// TIA Portal V17 export
// export: Created 2025-06-26T07:49:16.3730664Z, ExportSetting WithDefaults, DisplayName Totally Integrated Automation Portal, DisplayVersion V17 Update 8, DisplayName TIA Portal Openness, DisplayVersion V17 Update 8, DisplayName TIA Portal Version Control Interface, DisplayVersion V17, DisplayName STEP 7 Professional, DisplayVersion V17 Update 8, DisplayName STEP 7 Safety, DisplayVersion V17 Update 6, DisplayName WinCC Advanced, DisplayVersion V17 Update 8
FUNCTION_BLOCK "CustomerInputProcessing"   // FB6, FBD
TITLE = Internalize customer values
{ S7_Optimized_Access := 'TRUE' }
AUTHOR : Heaten
VERSION : 0.1
// stored: AutoNumber true, IsIECCheckEnabled false, IsRetainMemResEnabled false, MemoryReserve 0, SetENOAutomatically false, UDAEnableTagReadback false
   VAR_INPUT
      bEnable : Bool;
   END_VAR
   VAR
      Dummy : Bool;
   END_VAR
BEGIN

REGION Network 1: Customer comm ok
END_REGION

REGION Network 2: Do processing or not
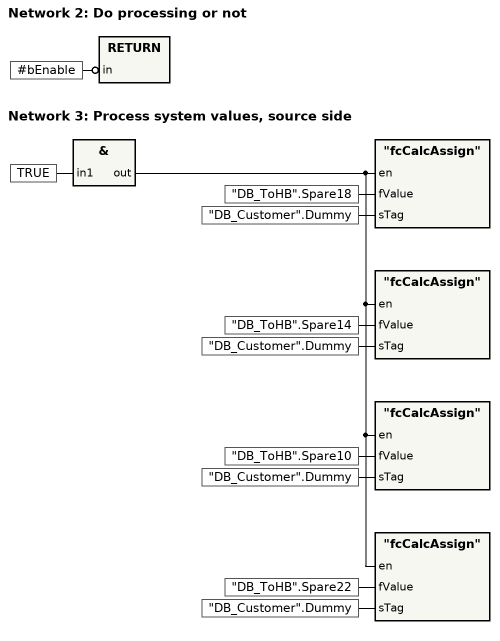
   IF NOT #bEnable THEN
       ENO := TRUE;
       RETURN;
   END_IF;
END_REGION

REGION Network 3: Process system values, source side
   IF TRUE THEN
       "fcCalcAssign"(fValue := "DB_ToHB".Spare18, sTag := "DB_Customer".Dummy);
       "fcCalcAssign"(fValue := "DB_ToHB".Spare14, sTag := "DB_Customer".Dummy);
       "fcCalcAssign"(fValue := "DB_ToHB".Spare10, sTag := "DB_Customer".Dummy);
       "fcCalcAssign"(fValue := "DB_ToHB".Spare22, sTag := "DB_Customer".Dummy);
   END_IF;
END_REGION

REGION Network 4: Beneo process system values, sink side
   // Including dryer air temperatures & Hall ambient measurements
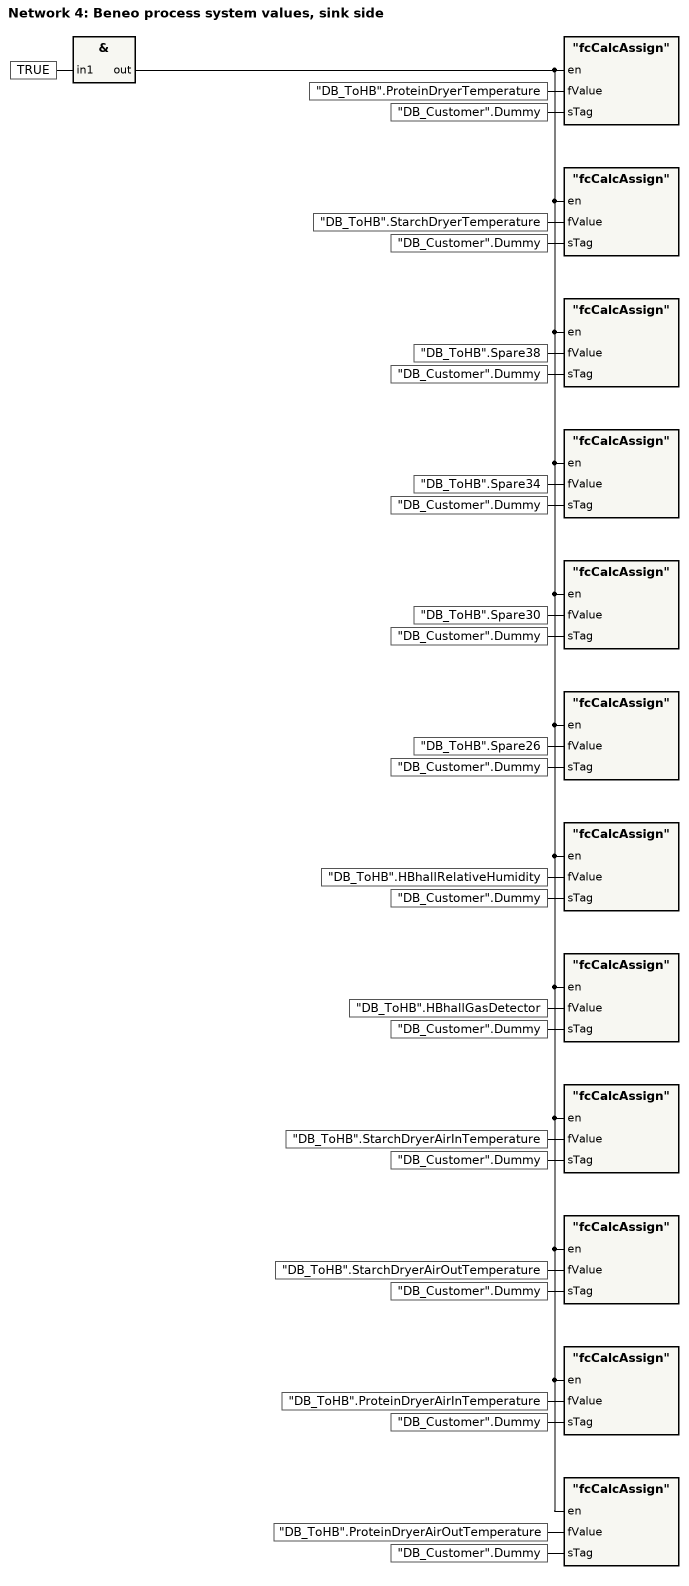
   IF TRUE THEN
       "fcCalcAssign"(fValue := "DB_ToHB".ProteinDryerTemperature, sTag := "DB_Customer".Dummy);
       "fcCalcAssign"(fValue := "DB_ToHB".StarchDryerTemperature, sTag := "DB_Customer".Dummy);
       "fcCalcAssign"(fValue := "DB_ToHB".Spare38, sTag := "DB_Customer".Dummy);
       "fcCalcAssign"(fValue := "DB_ToHB".Spare34, sTag := "DB_Customer".Dummy);
       "fcCalcAssign"(fValue := "DB_ToHB".Spare30, sTag := "DB_Customer".Dummy);
       "fcCalcAssign"(fValue := "DB_ToHB".Spare26, sTag := "DB_Customer".Dummy);
       "fcCalcAssign"(fValue := "DB_ToHB".HBhallRelativeHumidity, sTag := "DB_Customer".Dummy);
       "fcCalcAssign"(fValue := "DB_ToHB".HBhallGasDetector, sTag := "DB_Customer".Dummy);
       "fcCalcAssign"(fValue := "DB_ToHB".StarchDryerAirInTemperature, sTag := "DB_Customer".Dummy);
       "fcCalcAssign"(fValue := "DB_ToHB".StarchDryerAirOutTemperature, sTag := "DB_Customer".Dummy);
       "fcCalcAssign"(fValue := "DB_ToHB".ProteinDryerAirInTemperature, sTag := "DB_Customer".Dummy);
       "fcCalcAssign"(fValue := "DB_ToHB".ProteinDryerAirOutTemperature, sTag := "DB_Customer".Dummy);
   END_IF;
END_REGION

REGION Network 5: Flow detection
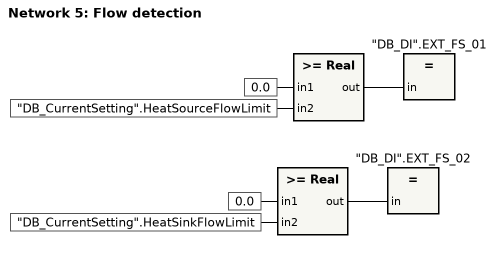
   "DB_DI".EXT_FS_01 := 0.0 >= "DB_CurrentSetting".HeatSourceFlowLimit;
   "DB_DI".EXT_FS_02 := 0.0 >= "DB_CurrentSetting".HeatSinkFlowLimit;
END_REGION
END_FUNCTION_BLOCK
